// TIA Portal project "yolcu otobüsü" (V16)

(* hardware
DEVICE "HMI_1"  KTP900 Basic PN
   slot 0: "HMI_1"  KTP900 Basic PN  6AV2 123-2JB03-0AX0  16.0.0.0
   slot 1: "HMI_RT_1"  KTP900 Basic PN  6AV2 123-2JB03-0AX0  16.0.0.0
   slot 5: "HMI_1.IE_CP_1"  PROFINET Interface  16.0.0.0
      slot 1: "PROFINET Interface_1"  PROFINET Interface
         slot 1: "Port_1"  Port
DEVICE "S71500/ET200MP station_1"  S7-1500 station
   slot 0: "Rail_0"  Rack  6ES7 590-1***0-0AA0
   slot 1: "PLC_1"  CPU 1515-2 PN  6ES7 515-2AM00-0AB0  V1.8
      slot 3: "CPU display_1"  6ES7591-1BA00-0AA0
      slot 32768: "PROFINET interface_1"  X1
         slot 32769: "Port_1"  X1 P1
         slot 32770: "Port_2"  X1 P2
      slot 33024: "PROFINET interface_2"  X2
         slot 33025: "Port_1"  X2 P1
*)

// ===== PLC "PLC_1"  CPU 1515-2 PN =====

VAR_GLOBAL   // PLC tag table "Default tag table"
   "İkaz Lambası" AT %M0.0 : Bool;
   "Açma-Kapama" AT %M0.1 : Bool;
   "Durdurma-1" AT %M0.2 : Bool;
   "Durdurma-2" AT %M0.3 : Bool;
   "Durdurma-3" AT %M0.4 : Bool;
   "Durdurma-4" AT %M0.5 : Bool;
   "Durdurma-5" AT %M0.6 : Bool;
   "Durdurma-6" AT %M0.7 : Bool;
   "Buzzer Aktif" AT %M1.0 : Bool;
   "Kapı sensörü" AT %M1.1 : Bool;
   "P_TRIG2" AT %M1.2 : Bool;
END_VAR

ORGANIZATION_BLOCK "Main"   // OB1, LAD, ProgramCycle
TITLE = "Main Program Sweep (Cycle)"
{ S7_Optimized_Access := 'TRUE' }
VERSION : 0.1
   VAR_INPUT
      Initial_Call : Bool;   // Initial call of this OB
      Remanence : Bool;   // =True, if remanent data are available
   END_VAR
   VAR_TEMP
      P_TRIG1 : Bool;
   END_VAR
   VAR_TEMP   // added for the SCL form of the ladder/FBD networks
      _w1 : Bool;
      _w2 : Bool;
      _w3 : Bool;
   END_VAR
BEGIN

REGION Network 1
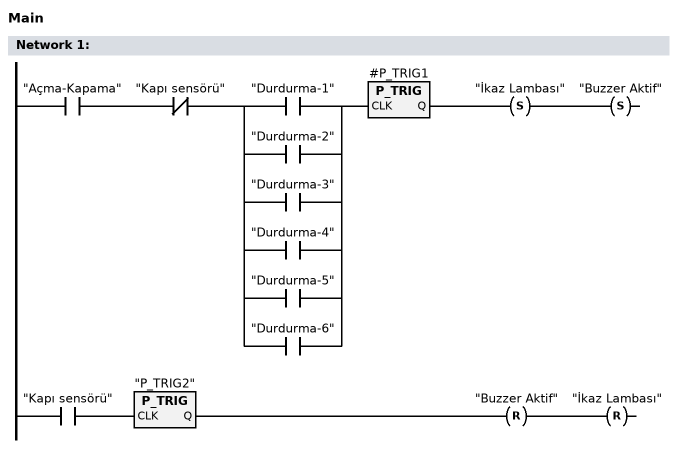
   RUNG wire#powerrail
      Contact( "Açma-Kapama" )
      I_Contact( "Kapı sensörü" )
      wire#w1
      Contact( "Durdurma-1" )
      wire#w2
      P_Trig( #P_TRIG1 )
      S_Coil( "İkaz Lambası" )
      S_Coil( "Buzzer Aktif" )
   END_RUNG
   RUNG wire#w1
      Contact( "Durdurma-2" )
   END_RUNG wire#w2
   RUNG wire#w1
      Contact( "Durdurma-3" )
   END_RUNG wire#w2
   RUNG wire#w1
      Contact( "Durdurma-4" )
   END_RUNG wire#w2
   RUNG wire#w1
      Contact( "Durdurma-5" )
   END_RUNG wire#w2
   RUNG wire#w1
      Contact( "Durdurma-6" )
   END_RUNG wire#w2
   RUNG wire#powerrail
      Contact( "Kapı sensörü" )
      P_Trig( "P_TRIG2" )
      R_Coil( "Buzzer Aktif" )
      R_Coil( "İkaz Lambası" )
   END_RUNG
   // the same network as SCL:
   #_w1 := "Açma-Kapama" AND NOT "Kapı sensörü" AND ("Durdurma-1" OR "Durdurma-2" OR "Durdurma-3" OR "Durdurma-4" OR "Durdurma-5" OR "Durdurma-6");
   #_w2 := #_w1 AND NOT #P_TRIG1;   // rising edge
   #P_TRIG1 := #_w1;
   IF #_w2 THEN
       "İkaz Lambası" := TRUE;
       "Buzzer Aktif" := TRUE;
   END_IF;
   #_w3 := "Kapı sensörü" AND NOT "P_TRIG2";   // rising edge
   "P_TRIG2" := "Kapı sensörü";
   IF #_w3 THEN
       "Buzzer Aktif" := FALSE;
       "İkaz Lambası" := FALSE;
   END_IF;
END_REGION
END_ORGANIZATION_BLOCK

(* ===== HMI "HMI_RT_1" =====
system functions are stored by id; their names below are inferred from use
connection "HMI_Connection_1": ETHERNET, SMART_S7_1500_OMS

HMI tags "Default tag table"
   "Tag_ScreenNumber" : UInt, internal
   "Açma-Kapama" : Bool = PLC "Açma-Kapama" AT %M0.1, 1 s
   "Buzzer Aktif" : Bool = PLC "Buzzer Aktif" AT %M1.0, 1 s
   "İkaz Lambası" : Bool = PLC "İkaz Lambası" AT %M0.0, 1 s
   "Kapı sensörü" : Bool = PLC "Kapı sensörü" AT %M1.1, 1 s
   "Durdurma-1" : Bool = PLC "Durdurma-1" AT %M0.2, 1 s
   "Durdurma-2" : Bool = PLC "Durdurma-2" AT %M0.3, 1 s
   "Durdurma-3" : Bool = PLC "Durdurma-3" AT %M0.4, 1 s
   "Durdurma-4" : Bool = PLC "Durdurma-4" AT %M0.5, 1 s
   "Durdurma-5" : Bool = PLC "Durdurma-5" AT %M0.6, 1 s
   "Durdurma-6" : Bool = PLC "Durdurma-6" AT %M0.7, 1 s

Template "Template_1" 800x480
   Button "Exit" at 722,440 size 55x39; TextOff 'Exit'; PictureOff "ExitRuntime_KTP900_Basic_PN_TR"; PictureOn "ExitRuntime_KTP900_Basic_PN_TR"
      on Release: StopRuntime(0)
   Button "Template_Button" at 622,440 size 55x39; TextOff 'Text'
   Button "Template_Button_1" at 522,440 size 55x39; TextOff 'Text'
   Button "Template_Button_2" at 422,440 size 55x39; TextOff 'Text'
   Button "Template_Button_3" at 322,440 size 55x39; TextOff 'Text'
   Button "Template_Button_4" at 222,440 size 55x39; TextOff 'Text'
   Button "Template_Button_5" at 122,440 size 55x39; TextOff 'Text'
   Button "Start screen" at 22,440 size 55x39; TextOff 'Start screen'; PictureOff "NavigateHome_KTP900_Basic_PN_TR"; PictureOn "NavigateHome_KTP900_Basic_PN_TR"
      on Release: ActivateScreen("Root screen", 0)
   SymbolicIOField "Symbolic_IO_Field_Screen" at 73,7 size 620x26; TextOff '0'; TextOn '1'; TextList "TextList_ScreenNames"
      ProcessValue <- "Tag_ScreenNumber"
      on Change: ActivateScreenByNumber("Tag_ScreenNumber", 0)
   DateTimeField "HmiScreenItemData" at 695,20 size 105x20
   DateTimeField "HmiScreenItemData_1" at 695,0 size 105x20
   GraphicView "Logo" at 0,0 size 71x40; Picture "Logo of HMI_1"

screen "Root screen" 800x480, template "Template_1"
   on GenerateScreen: SetTag("Tag_ScreenNumber", 1)
   TextField "Text field_1" at 83,97 size 14x20; Text 'Text'
   Button "Button_1" at 36,65 size 96x32; TextOff 'Açma-Kapama'
      on Press: InvertBit("Açma-Kapama")
   TextField "Text field_2" at 285,65 size 93x20; Text 'Buzzer Aktif :'
   Circle "Circle_1" at 402,50 size 48x48
      Appearance <- "Buzzer Aktif"
   TextField "Text field_3" at 285,132 size 93x20; Text 'İkaz Lambası:'
   Circle "Circle_2" at 402,117 size 48x48
      Appearance <- "İkaz Lambası"
   Button "Button_2" at 36,163 size 96x32; TextOff 'Kapı Sensörü'
      on Press: InvertBit("Kapı sensörü")
   Button "Button_3" at 37,215 size 96x32; TextOff 'Durdur-1'
      on Press: InvertBit("Durdurma-1")
   Button "Button_4" at 37,258 size 96x32; TextOff 'Durdur-2'
      on Press: InvertBit("Durdurma-2")
   Button "Button_5" at 37,307 size 96x32; TextOff 'Durdur-3'
      on Press: InvertBit("Durdurma-3")
   Button "Button_6" at 36,347 size 96x32; TextOff 'Durdur-4'
      on Press: InvertBit("Durdurma-4")
   Button "Button_7" at 36,388 size 96x32; TextOff 'Durdur-5'
      on Press: InvertBit("Durdurma-5")
   Button "Button_8" at 36,426 size 96x32; TextOff 'Durdur-6'
      on Press: InvertBit("Durdurma-6")
   Circle "Circle_10" at 148,59 size 38x38
      Appearance <- "Açma-Kapama"
   Circle "Circle_3" at 147,157 size 38x38
      Appearance <- "Kapı sensörü"
   Circle "Circle_4" at 149,252 size 38x38
      Appearance <- "Durdurma-2"
   Circle "Circle_5" at 148,205 size 38x38
      Appearance <- "Durdurma-1"
   Circle "Circle_6" at 149,301 size 38x38
      Appearance <- "Durdurma-3"
   Circle "Circle_7" at 150,386 size 38x38
      Appearance <- "Durdurma-5"
   Circle "Circle_8" at 149,347 size 38x38
      Appearance <- "Durdurma-4"
   Circle "Circle_9" at 152,426 size 38x38
      Appearance <- "Durdurma-6"
*)